VAR_GLOBAL CONSTANT
	receiveBufferSize : UINT := 2048;
	TimeOut : TIME := T#25S;
	MAX_TASK_SIZE : UINT := 20;
END_VAR

(* stored: Version 1.1.0.1
   GVL RoboConnectParams: Id {c8eefda0-577a-4804-a57d-129301a69a2f}, ParameterList True *)
